(* PLC project Unnamed, Unknown Unnamed 1 *)
(* stored: creationDateTime 2025-06-04T18:25:43, modificationDateTime 2025-06-04T19:16:09 *)

PROGRAM part_1a
  VAR
    Input0 AT %IX1.0 : BOOL;
    Input1 AT %IX1.1 : BOOL;
    Output0 AT %QX1.0 : BOOL;
    Output1 AT %QX1.1 : BOOL;
  END_VAR
  VAR
    TP0 : TP;
  END_VAR

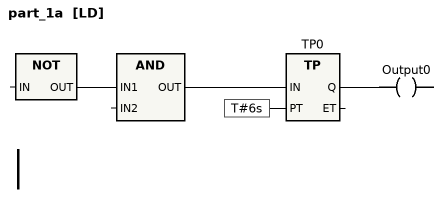
(* LD diagram, written out as Structured Text *)
TP0(IN := AND(IN1 := NOT()), PT := T#6s);
Output0 := TP0.Q;
END_PROGRAM

CONFIGURATION Config0
  RESOURCE Res0 ON PLC
    TASK task0(INTERVAL := T#20ms, PRIORITY := 0);
    PROGRAM instance0 WITH task0 : part_1a;
  END_RESOURCE
END_CONFIGURATION
